// TIA Portal V21 export
DATA_BLOCK "BatchTimer"   // DB315
{ S7_Optimized_Access := 'TRUE' }
// stored: AutoNumber false, MemoryReserve 100
   VAR
      Timer01 : IEC_TIMER;
      Timer02 { S7_SetPoint := 'True'} : IEC_TIMER;
      Timer03 { S7_SetPoint := 'True'} : IEC_TIMER;
      Timer04 { S7_SetPoint := 'True'} : IEC_TIMER;
      Timer05 { S7_SetPoint := 'True'} : IEC_TIMER;
      Timer06 { S7_SetPoint := 'True'} : IEC_TIMER;
      Timer07 { S7_SetPoint := 'True'} : IEC_TIMER;
      Timer08 { S7_SetPoint := 'True'} : IEC_TIMER;
      Timer09 { S7_SetPoint := 'True'} : IEC_TIMER;
      Timer10 { S7_SetPoint := 'True'} : IEC_TIMER;
      Timer11 { S7_SetPoint := 'True'} : IEC_TIMER;
      Timer12 { S7_SetPoint := 'True'} : IEC_TIMER;
      Timer13 { S7_SetPoint := 'True'} : IEC_TIMER;
      Timer14 { S7_SetPoint := 'True'} : IEC_TIMER;
      Timer15 { S7_SetPoint := 'True'} : IEC_TIMER;
      Timer16 { S7_SetPoint := 'True'} : IEC_TIMER;
      Timer17 { S7_SetPoint := 'True'} : IEC_TIMER;
      Timer18 { S7_SetPoint := 'True'} : IEC_TIMER;
      Timer19 { S7_SetPoint := 'True'} : IEC_TIMER;
      Timer20 { S7_SetPoint := 'True'} : IEC_TIMER;
      Timer21 { S7_SetPoint := 'True'} : IEC_TIMER;
      Timer22 { S7_SetPoint := 'True'} : IEC_TIMER;
      Timer23 { S7_SetPoint := 'True'} : IEC_TIMER;
      Timer24 { S7_SetPoint := 'True'} : IEC_TIMER;
      Timer25 { S7_SetPoint := 'True'} : IEC_TIMER;
      Timer26 { S7_SetPoint := 'True'} : IEC_TIMER;
      Timer27 { S7_SetPoint := 'True'} : IEC_TIMER;
      Timer28 { S7_SetPoint := 'True'} : IEC_TIMER;
      Timer29 { S7_SetPoint := 'True'} : IEC_TIMER;
      Timer30 { S7_SetPoint := 'True'} : IEC_TIMER;
      Timer31 { S7_SetPoint := 'True'} : IEC_TIMER;
      Timer32 { S7_SetPoint := 'True'} : IEC_TIMER;
      Timer33 { S7_SetPoint := 'True'} : IEC_TIMER;
      Timer34 { S7_SetPoint := 'True'} : IEC_TIMER;
      Timer35 { S7_SetPoint := 'True'} : IEC_TIMER;
      Timer36 { S7_SetPoint := 'True'} : IEC_TIMER;
      Timer37 { S7_SetPoint := 'True'} : IEC_TIMER;
      Timer38 { S7_SetPoint := 'True'} : IEC_TIMER;
      Timer39 { S7_SetPoint := 'True'} : IEC_TIMER;
      Timer40 { S7_SetPoint := 'True'} : IEC_TIMER;
      Timer41 { S7_SetPoint := 'True'} : IEC_TIMER;
      Timer42 { S7_SetPoint := 'True'} : IEC_TIMER;
      Timer43 { S7_SetPoint := 'True'} : IEC_TIMER;
      Timer44 { S7_SetPoint := 'True'} : IEC_TIMER;
      Timer45 { S7_SetPoint := 'True'} : IEC_TIMER;
      Timer46 { S7_SetPoint := 'True'} : IEC_TIMER;
      Timer47 { S7_SetPoint := 'True'} : IEC_TIMER;
      Timer48 { S7_SetPoint := 'True'} : IEC_TIMER;
      Timer49 { S7_SetPoint := 'True'} : IEC_TIMER;
      Timer50 { S7_SetPoint := 'True'} : IEC_TIMER;
      Timer51 { S7_SetPoint := 'True'} : IEC_TIMER;
      Timer52 { S7_SetPoint := 'True'} : IEC_TIMER;
      Timer53 { S7_SetPoint := 'True'} : IEC_TIMER;
      Timer54 { S7_SetPoint := 'True'} : IEC_TIMER;
      Timer55 { S7_SetPoint := 'True'} : IEC_TIMER;
      Timer56 { S7_SetPoint := 'True'} : IEC_TIMER;
      Timer57 { S7_SetPoint := 'True'} : IEC_TIMER;
      Timer58 { S7_SetPoint := 'True'} : IEC_TIMER;
      Timer59 { S7_SetPoint := 'True'} : IEC_TIMER;
      Timer60 { S7_SetPoint := 'True'} : IEC_TIMER;
      Timer61 { S7_SetPoint := 'True'} : IEC_TIMER;
      Timer62 { S7_SetPoint := 'True'} : IEC_TIMER;
      Timer63 { S7_SetPoint := 'True'} : IEC_TIMER;
      Timer64 { S7_SetPoint := 'True'} : IEC_TIMER;
      Timer65 { S7_SetPoint := 'True'} : IEC_TIMER;
   END_VAR
BEGIN
END_DATA_BLOCK
